// TIA Portal V17 export
// export: Created 2023-02-13T11:16:32.2818041Z, ExportSetting WithDefaults, DisplayName Totally Integrated Automation Portal, DisplayVersion V17, DisplayName TIA Portal Openness, DisplayVersion V17, DisplayName TIA Portal Teamcenter Gateway, DisplayVersion V17, DisplayName TIA Portal Version Control Interface, DisplayVersion V17, DisplayName SINAMICS Startdrive Advanced, DisplayVersion V17, DisplayName SINAMICS Startdrive G130, G150, S120, S150, SINAMICS MV, S210, DisplayVersion V17, DisplayName SINAMICS Startdrive G110M, G120, G120C, G120D, G120P, G115D, DisplayVersion V17, DisplayName STEP 7 Professional, DisplayVersion V17, DisplayName STEP 7 Safety, DisplayVersion V17, DisplayName WinCC Professional, DisplayVersion V17
FUNCTION_BLOCK "IO Valve T51 HotWaterLine"   // FB311, LAD
{ S7_Optimized_Access := 'FALSE' }
VERSION : 0.1
// stored: AutoNumber false, IsIECCheckEnabled false, SetENOAutomatically false, UDAEnableTagReadback false
   VAR_INPUT
      lock : Bool;
      Init : Bool;
      testing : Bool;
      Reset : Bool;
   END_VAR
   VAR
      "AV-51.01" { S7_SetPoint := 'True'} : "Valve";
      "AV-51.02" { S7_SetPoint := 'True'} : "Valve";
      "AV-51.03" { S7_SetPoint := 'True'} : "Valve";
      "AV-51.04" { S7_SetPoint := 'True'} : "Valve";
      "AV-51.05" { S7_SetPoint := 'True'} : "Valve";
      "AV-51.06" { S7_SetPoint := 'True'} : "Valve";
      "AV-51.07" { S7_SetPoint := 'True'} : "Valve";
      "AV-51.08" { S7_SetPoint := 'True'} : "Valve";
      "AV-51.09" { S7_SetPoint := 'True'} : "Valve";
      "AV-51.10" { S7_SetPoint := 'True'} : "Valve";
      "AV-51.11" { S7_SetPoint := 'True'} : "Valve";
      "AV-51.12" { S7_SetPoint := 'True'} : "Valve";
      "AV-51.13" { S7_SetPoint := 'True'} : "Valve";
      "AV-51.14" { S7_SetPoint := 'True'} : "Valve";
      "AV-51.15" { S7_SetPoint := 'True'} : "Valve";
      "CV-51.11" { S7_SetPoint := 'True'} : "Valve";
   END_VAR
BEGIN

REGION Network 1 (SCL): FB OPEN and CLOSE
   IF #testing THEN
       // Statement section IF
       #"AV-51.01".FB_OPEN := #"AV-51.01".QCMD_OP;
       #"AV-51.01".FB_CLOSE := NOT #"AV-51.01".QCMD_OP;
       #"AV-51.02".FB_OPEN := #"AV-51.02".QCMD_OP;
       #"AV-51.02".FB_CLOSE := NOT #"AV-51.02".QCMD_OP;
       #"AV-51.03".FB_OPEN := #"AV-51.03".QCMD_OP;
       #"AV-51.03".FB_CLOSE := NOT #"AV-51.03".QCMD_OP;
       #"AV-51.04".FB_OPEN := #"AV-51.04".QCMD_OP;
       #"AV-51.04".FB_CLOSE := NOT #"AV-51.04".QCMD_OP;
       #"AV-51.05".FB_OPEN := #"AV-51.05".QCMD_OP;
       #"AV-51.05".FB_CLOSE := NOT #"AV-51.05".QCMD_OP;
       #"AV-51.06".FB_OPEN := #"AV-51.06".QCMD_OP;
       #"AV-51.06".FB_CLOSE := NOT #"AV-51.06".QCMD_OP;
       #"AV-51.07".FB_OPEN := #"AV-51.07".QCMD_OP;
       #"AV-51.07".FB_CLOSE := NOT #"AV-51.07".QCMD_OP;
       #"AV-51.08".FB_OPEN := #"AV-51.08".QCMD_OP;
       #"AV-51.08".FB_CLOSE := NOT #"AV-51.08".QCMD_OP;
       #"AV-51.09".FB_OPEN := #"AV-51.09".QCMD_OP;
       #"AV-51.09".FB_CLOSE := NOT #"AV-51.09".QCMD_OP;
       #"AV-51.10".FB_OPEN := #"AV-51.10".QCMD_OP;
       #"AV-51.10".FB_CLOSE := NOT #"AV-51.10".QCMD_OP;
       #"AV-51.11".FB_OPEN := #"AV-51.11".QCMD_OP;
       #"AV-51.11".FB_CLOSE := NOT #"AV-51.11".QCMD_OP;
       #"AV-51.12".FB_OPEN := #"AV-51.12".QCMD_OP;
       #"AV-51.12".FB_CLOSE := NOT #"AV-51.12".QCMD_OP;
       #"AV-51.13".FB_OPEN := #"AV-51.13".QCMD_OP;
       #"AV-51.13".FB_CLOSE := NOT #"AV-51.13".QCMD_OP;
       #"AV-51.14".FB_OPEN := #"AV-51.14".QCMD_OP;
       #"AV-51.14".FB_CLOSE := NOT #"AV-51.14".QCMD_OP;
       #"AV-51.15".FB_OPEN := #"AV-51.15".QCMD_OP;
       #"AV-51.15".FB_CLOSE := NOT #"AV-51.15".QCMD_OP;
   ELSE
       // Statement section ELSE
       #"AV-51.01".FB_OPEN := #"AV-51.01".QCMD_OP;
       #"AV-51.01".FB_CLOSE := NOT #"AV-51.01".QCMD_OP;
       #"AV-51.02".FB_OPEN := #"AV-51.02".QCMD_OP;
       #"AV-51.02".FB_CLOSE := NOT #"AV-51.02".QCMD_OP;
       #"AV-51.03".FB_OPEN := #"AV-51.03".QCMD_OP;
       #"AV-51.03".FB_CLOSE := NOT #"AV-51.03".QCMD_OP;
       #"AV-51.04".FB_OPEN := NOT "ZSC-51.04";
       #"AV-51.04".FB_CLOSE := "ZSC-51.04";
       #"AV-51.05".FB_OPEN := NOT "ZSC-51.05";
       #"AV-51.05".FB_CLOSE := "ZSC-51.05";
       #"AV-51.06".FB_OPEN := #"AV-51.06".QCMD_OP;
       #"AV-51.06".FB_CLOSE := NOT #"AV-51.06".QCMD_OP;
       #"AV-51.07".FB_OPEN := #"AV-51.07".QCMD_OP;
       #"AV-51.07".FB_CLOSE := NOT #"AV-51.07".QCMD_OP;
       #"AV-51.08".FB_OPEN := #"AV-51.08".QCMD_OP;
       #"AV-51.08".FB_CLOSE := NOT #"AV-51.08".QCMD_OP;
       #"AV-51.09".FB_OPEN := #"AV-51.09".QCMD_OP;
       #"AV-51.09".FB_CLOSE := NOT #"AV-51.09".QCMD_OP;
       #"AV-51.10".FB_OPEN := #"AV-51.10".QCMD_OP;
       #"AV-51.10".FB_CLOSE := NOT #"AV-51.10".QCMD_OP;
       #"AV-51.11".FB_OPEN := #"AV-51.11".QCMD_OP;
       #"AV-51.11".FB_CLOSE := NOT #"AV-51.11".QCMD_OP;
       #"AV-51.12".FB_OPEN := #"AV-51.12".QCMD_OP;
       #"AV-51.12".FB_CLOSE := NOT #"AV-51.12".QCMD_OP;
       #"AV-51.13".FB_OPEN := #"AV-51.13".QCMD_OP;
       #"AV-51.13".FB_CLOSE := NOT #"AV-51.13".QCMD_OP;
       #"AV-51.14".FB_OPEN := #"AV-51.14".QCMD_OP;
       #"AV-51.14".FB_CLOSE := NOT #"AV-51.14".QCMD_OP;
       #"AV-51.15".FB_OPEN := #"AV-51.15".QCMD_OP;
       #"AV-51.15".FB_CLOSE := NOT #"AV-51.15".QCMD_OP;
   END_IF;
END_REGION

NETWORK
TITLE = FB Monitoring Time
// FB OPEN Time
      L     t#20s;
      T     #"AV-51.01".MON_T;
      T     #"AV-51.02".MON_T;
      T     #"AV-51.03".MON_T;
      T     #"AV-51.04".MON_T;
      T     #"AV-51.05".MON_T;
      T     #"AV-51.06".MON_T;
      T     #"AV-51.07".MON_T;
      T     #"AV-51.08".MON_T;
      T     #"AV-51.09".MON_T;
      T     #"AV-51.10".MON_T;
      T     #"AV-51.11".MON_T;
      T     #"AV-51.12".MON_T;
      T     #"AV-51.13".MON_T;
      T     #"AV-51.14".MON_T;
      T     #"AV-51.15".MON_T;
// FB CLOSE Time
      L     t#20s;
      T     #"AV-51.01".MON_T_CLOSE;
      T     #"AV-51.02".MON_T_CLOSE;
      T     #"AV-51.03".MON_T_CLOSE;
      T     #"AV-51.04".MON_T_CLOSE;
      T     #"AV-51.05".MON_T_CLOSE;
      T     #"AV-51.06".MON_T_CLOSE;
      T     #"AV-51.07".MON_T_CLOSE;
      T     #"AV-51.08".MON_T_CLOSE;
      T     #"AV-51.09".MON_T_CLOSE;
      T     #"AV-51.10".MON_T_CLOSE;
      T     #"AV-51.11".MON_T_CLOSE;
      T     #"AV-51.12".MON_T_CLOSE;
      T     #"AV-51.13".MON_T_CLOSE;
      T     #"AV-51.14".MON_T_CLOSE;
      T     #"AV-51.15".MON_T_CLOSE;

REGION Network 3: AV-51.01
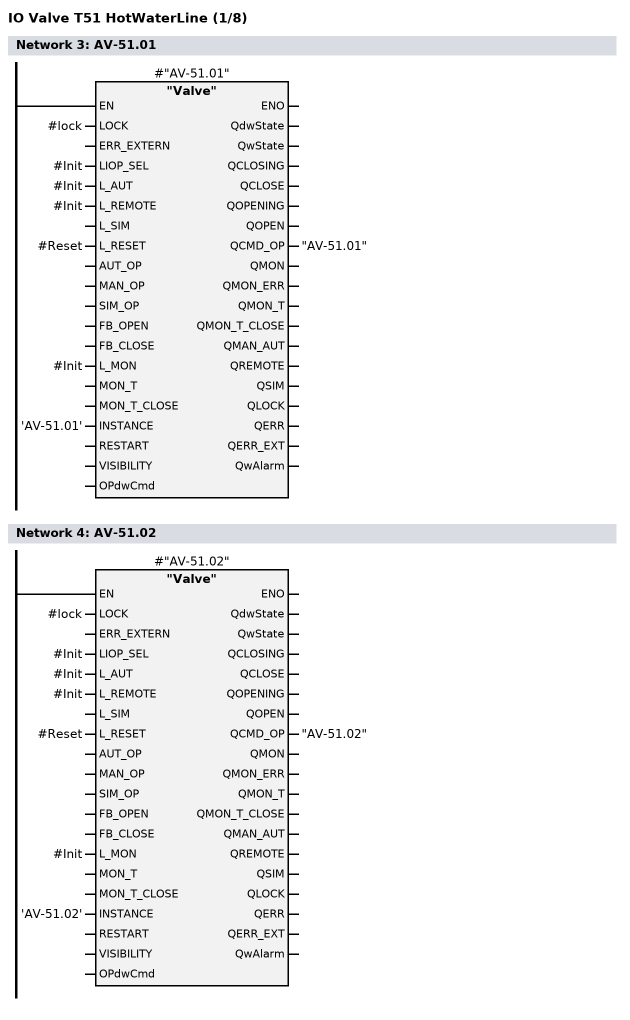
   RUNG wire#powerrail
      #"AV-51.01"(LOCK := #lock, ERR_EXTERN :=, LIOP_SEL := #Init, L_AUT := #Init, L_REMOTE := #Init, L_SIM :=, L_RESET := #Reset, AUT_OP :=, MAN_OP :=, SIM_OP :=, FB_OPEN :=, FB_CLOSE :=, L_MON := #Init, MON_T :=, MON_T_CLOSE :=, INSTANCE := 'AV-51.01', RESTART :=, VISIBILITY :=, OPdwCmd :=, QdwState =>, QwState =>, QCLOSING =>, QCLOSE =>, QOPENING =>, QOPEN =>, QCMD_OP => "AV-51.01", QMON =>, QMON_ERR =>, QMON_T =>, QMON_T_CLOSE =>, QMAN_AUT =>, QREMOTE =>, QSIM =>, QLOCK =>, QERR =>, QERR_EXT =>, QwAlarm =>)
   END_RUNG
   // the same network as SCL:
   #"AV-51.01"(LOCK := #lock,   // "Valve"
               LIOP_SEL := #Init,
               L_AUT := #Init,
               L_REMOTE := #Init,
               L_RESET := #Reset,
               L_MON := #Init,
               INSTANCE := 'AV-51.01',
               QCMD_OP => "AV-51.01");
END_REGION

REGION Network 4: AV-51.02
   RUNG wire#powerrail
      #"AV-51.02"(LOCK := #lock, ERR_EXTERN :=, LIOP_SEL := #Init, L_AUT := #Init, L_REMOTE := #Init, L_SIM :=, L_RESET := #Reset, AUT_OP :=, MAN_OP :=, SIM_OP :=, FB_OPEN :=, FB_CLOSE :=, L_MON := #Init, MON_T :=, MON_T_CLOSE :=, INSTANCE := 'AV-51.02', RESTART :=, VISIBILITY :=, OPdwCmd :=, QdwState =>, QwState =>, QCLOSING =>, QCLOSE =>, QOPENING =>, QOPEN =>, QCMD_OP => "AV-51.02", QMON =>, QMON_ERR =>, QMON_T =>, QMON_T_CLOSE =>, QMAN_AUT =>, QREMOTE =>, QSIM =>, QLOCK =>, QERR =>, QERR_EXT =>, QwAlarm =>)
   END_RUNG
   // the same network as SCL:
   #"AV-51.02"(LOCK := #lock,   // "Valve"
               LIOP_SEL := #Init,
               L_AUT := #Init,
               L_REMOTE := #Init,
               L_RESET := #Reset,
               L_MON := #Init,
               INSTANCE := 'AV-51.02',
               QCMD_OP => "AV-51.02");
END_REGION

REGION Network 5: AV-51.03
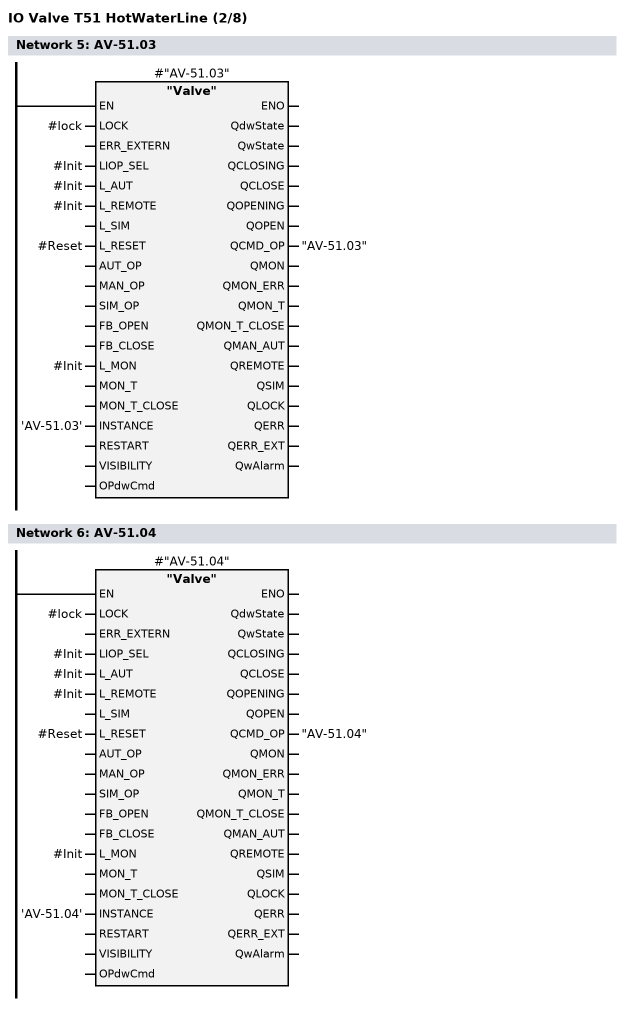
   RUNG wire#powerrail
      #"AV-51.03"(LOCK := #lock, ERR_EXTERN :=, LIOP_SEL := #Init, L_AUT := #Init, L_REMOTE := #Init, L_SIM :=, L_RESET := #Reset, AUT_OP :=, MAN_OP :=, SIM_OP :=, FB_OPEN :=, FB_CLOSE :=, L_MON := #Init, MON_T :=, MON_T_CLOSE :=, INSTANCE := 'AV-51.03', RESTART :=, VISIBILITY :=, OPdwCmd :=, QdwState =>, QwState =>, QCLOSING =>, QCLOSE =>, QOPENING =>, QOPEN =>, QCMD_OP => "AV-51.03", QMON =>, QMON_ERR =>, QMON_T =>, QMON_T_CLOSE =>, QMAN_AUT =>, QREMOTE =>, QSIM =>, QLOCK =>, QERR =>, QERR_EXT =>, QwAlarm =>)
   END_RUNG
   // the same network as SCL:
   #"AV-51.03"(LOCK := #lock,   // "Valve"
               LIOP_SEL := #Init,
               L_AUT := #Init,
               L_REMOTE := #Init,
               L_RESET := #Reset,
               L_MON := #Init,
               INSTANCE := 'AV-51.03',
               QCMD_OP => "AV-51.03");
END_REGION

REGION Network 6: AV-51.04
   RUNG wire#powerrail
      #"AV-51.04"(LOCK := #lock, ERR_EXTERN :=, LIOP_SEL := #Init, L_AUT := #Init, L_REMOTE := #Init, L_SIM :=, L_RESET := #Reset, AUT_OP :=, MAN_OP :=, SIM_OP :=, FB_OPEN :=, FB_CLOSE :=, L_MON := #Init, MON_T :=, MON_T_CLOSE :=, INSTANCE := 'AV-51.04', RESTART :=, VISIBILITY :=, OPdwCmd :=, QdwState =>, QwState =>, QCLOSING =>, QCLOSE =>, QOPENING =>, QOPEN =>, QCMD_OP => "AV-51.04", QMON =>, QMON_ERR =>, QMON_T =>, QMON_T_CLOSE =>, QMAN_AUT =>, QREMOTE =>, QSIM =>, QLOCK =>, QERR =>, QERR_EXT =>, QwAlarm =>)
   END_RUNG
   // the same network as SCL:
   #"AV-51.04"(LOCK := #lock,   // "Valve"
               LIOP_SEL := #Init,
               L_AUT := #Init,
               L_REMOTE := #Init,
               L_RESET := #Reset,
               L_MON := #Init,
               INSTANCE := 'AV-51.04',
               QCMD_OP => "AV-51.04");
END_REGION

REGION Network 7: AV-51.05
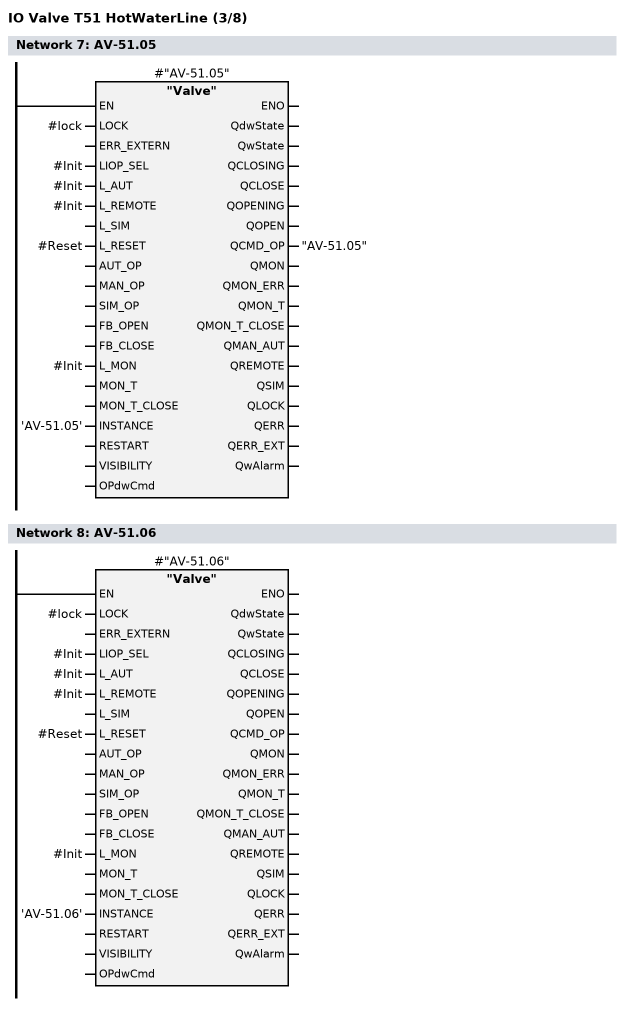
   RUNG wire#powerrail
      #"AV-51.05"(LOCK := #lock, ERR_EXTERN :=, LIOP_SEL := #Init, L_AUT := #Init, L_REMOTE := #Init, L_SIM :=, L_RESET := #Reset, AUT_OP :=, MAN_OP :=, SIM_OP :=, FB_OPEN :=, FB_CLOSE :=, L_MON := #Init, MON_T :=, MON_T_CLOSE :=, INSTANCE := 'AV-51.05', RESTART :=, VISIBILITY :=, OPdwCmd :=, QdwState =>, QwState =>, QCLOSING =>, QCLOSE =>, QOPENING =>, QOPEN =>, QCMD_OP => "AV-51.05", QMON =>, QMON_ERR =>, QMON_T =>, QMON_T_CLOSE =>, QMAN_AUT =>, QREMOTE =>, QSIM =>, QLOCK =>, QERR =>, QERR_EXT =>, QwAlarm =>)
   END_RUNG
   // the same network as SCL:
   #"AV-51.05"(LOCK := #lock,   // "Valve"
               LIOP_SEL := #Init,
               L_AUT := #Init,
               L_REMOTE := #Init,
               L_RESET := #Reset,
               L_MON := #Init,
               INSTANCE := 'AV-51.05',
               QCMD_OP => "AV-51.05");
END_REGION

REGION Network 8: AV-51.06
   RUNG wire#powerrail
      #"AV-51.06"(LOCK := #lock, ERR_EXTERN :=, LIOP_SEL := #Init, L_AUT := #Init, L_REMOTE := #Init, L_SIM :=, L_RESET := #Reset, AUT_OP :=, MAN_OP :=, SIM_OP :=, FB_OPEN :=, FB_CLOSE :=, L_MON := #Init, MON_T :=, MON_T_CLOSE :=, INSTANCE := 'AV-51.06', RESTART :=, VISIBILITY :=, OPdwCmd :=, QdwState =>, QwState =>, QCLOSING =>, QCLOSE =>, QOPENING =>, QOPEN =>, QCMD_OP =>, QMON =>, QMON_ERR =>, QMON_T =>, QMON_T_CLOSE =>, QMAN_AUT =>, QREMOTE =>, QSIM =>, QLOCK =>, QERR =>, QERR_EXT =>, QwAlarm =>)
   END_RUNG
   // the same network as SCL:
   #"AV-51.06"(LOCK := #lock,   // "Valve"
               LIOP_SEL := #Init,
               L_AUT := #Init,
               L_REMOTE := #Init,
               L_RESET := #Reset,
               L_MON := #Init,
               INSTANCE := 'AV-51.06');
END_REGION

REGION Network 9: AV-51.07
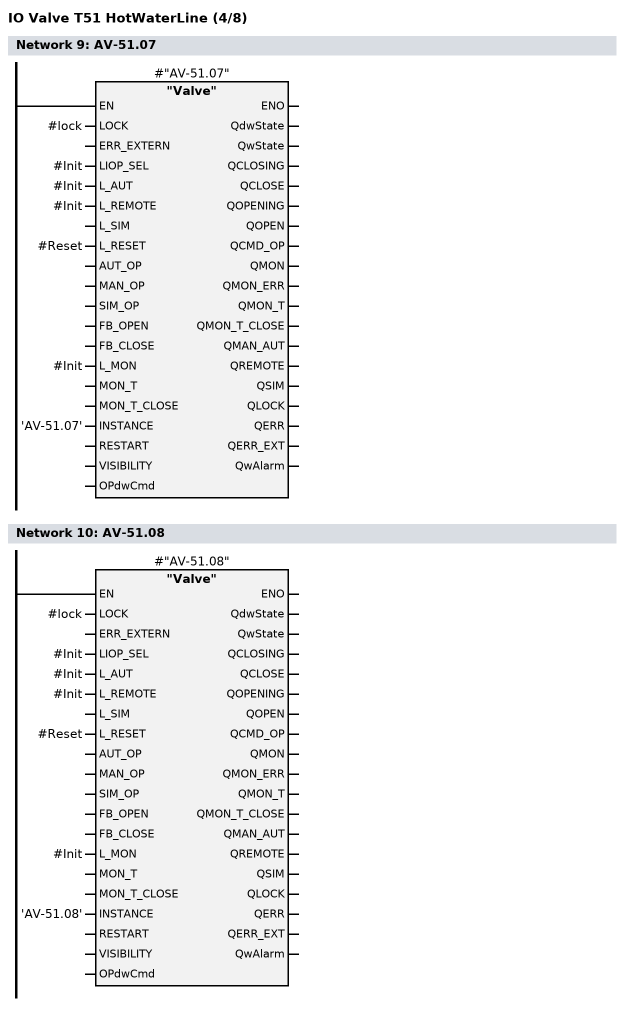
   RUNG wire#powerrail
      #"AV-51.07"(LOCK := #lock, ERR_EXTERN :=, LIOP_SEL := #Init, L_AUT := #Init, L_REMOTE := #Init, L_SIM :=, L_RESET := #Reset, AUT_OP :=, MAN_OP :=, SIM_OP :=, FB_OPEN :=, FB_CLOSE :=, L_MON := #Init, MON_T :=, MON_T_CLOSE :=, INSTANCE := 'AV-51.07', RESTART :=, VISIBILITY :=, OPdwCmd :=, QdwState =>, QwState =>, QCLOSING =>, QCLOSE =>, QOPENING =>, QOPEN =>, QCMD_OP =>, QMON =>, QMON_ERR =>, QMON_T =>, QMON_T_CLOSE =>, QMAN_AUT =>, QREMOTE =>, QSIM =>, QLOCK =>, QERR =>, QERR_EXT =>, QwAlarm =>)
   END_RUNG
   // the same network as SCL:
   #"AV-51.07"(LOCK := #lock,   // "Valve"
               LIOP_SEL := #Init,
               L_AUT := #Init,
               L_REMOTE := #Init,
               L_RESET := #Reset,
               L_MON := #Init,
               INSTANCE := 'AV-51.07');
END_REGION

REGION Network 10: AV-51.08
   RUNG wire#powerrail
      #"AV-51.08"(LOCK := #lock, ERR_EXTERN :=, LIOP_SEL := #Init, L_AUT := #Init, L_REMOTE := #Init, L_SIM :=, L_RESET := #Reset, AUT_OP :=, MAN_OP :=, SIM_OP :=, FB_OPEN :=, FB_CLOSE :=, L_MON := #Init, MON_T :=, MON_T_CLOSE :=, INSTANCE := 'AV-51.08', RESTART :=, VISIBILITY :=, OPdwCmd :=, QdwState =>, QwState =>, QCLOSING =>, QCLOSE =>, QOPENING =>, QOPEN =>, QCMD_OP =>, QMON =>, QMON_ERR =>, QMON_T =>, QMON_T_CLOSE =>, QMAN_AUT =>, QREMOTE =>, QSIM =>, QLOCK =>, QERR =>, QERR_EXT =>, QwAlarm =>)
   END_RUNG
   // the same network as SCL:
   #"AV-51.08"(LOCK := #lock,   // "Valve"
               LIOP_SEL := #Init,
               L_AUT := #Init,
               L_REMOTE := #Init,
               L_RESET := #Reset,
               L_MON := #Init,
               INSTANCE := 'AV-51.08');
END_REGION

REGION Network 11: AV-51.09
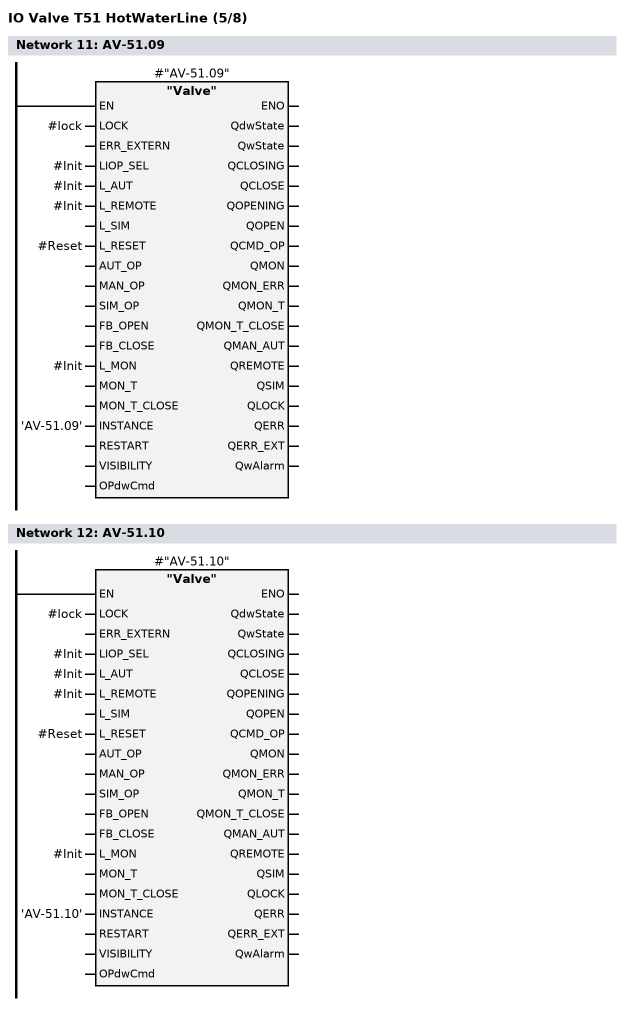
   RUNG wire#powerrail
      #"AV-51.09"(LOCK := #lock, ERR_EXTERN :=, LIOP_SEL := #Init, L_AUT := #Init, L_REMOTE := #Init, L_SIM :=, L_RESET := #Reset, AUT_OP :=, MAN_OP :=, SIM_OP :=, FB_OPEN :=, FB_CLOSE :=, L_MON := #Init, MON_T :=, MON_T_CLOSE :=, INSTANCE := 'AV-51.09', RESTART :=, VISIBILITY :=, OPdwCmd :=, QdwState =>, QwState =>, QCLOSING =>, QCLOSE =>, QOPENING =>, QOPEN =>, QCMD_OP =>, QMON =>, QMON_ERR =>, QMON_T =>, QMON_T_CLOSE =>, QMAN_AUT =>, QREMOTE =>, QSIM =>, QLOCK =>, QERR =>, QERR_EXT =>, QwAlarm =>)
   END_RUNG
   // the same network as SCL:
   #"AV-51.09"(LOCK := #lock,   // "Valve"
               LIOP_SEL := #Init,
               L_AUT := #Init,
               L_REMOTE := #Init,
               L_RESET := #Reset,
               L_MON := #Init,
               INSTANCE := 'AV-51.09');
END_REGION

REGION Network 12: AV-51.10
   RUNG wire#powerrail
      #"AV-51.10"(LOCK := #lock, ERR_EXTERN :=, LIOP_SEL := #Init, L_AUT := #Init, L_REMOTE := #Init, L_SIM :=, L_RESET := #Reset, AUT_OP :=, MAN_OP :=, SIM_OP :=, FB_OPEN :=, FB_CLOSE :=, L_MON := #Init, MON_T :=, MON_T_CLOSE :=, INSTANCE := 'AV-51.10', RESTART :=, VISIBILITY :=, OPdwCmd :=, QdwState =>, QwState =>, QCLOSING =>, QCLOSE =>, QOPENING =>, QOPEN =>, QCMD_OP =>, QMON =>, QMON_ERR =>, QMON_T =>, QMON_T_CLOSE =>, QMAN_AUT =>, QREMOTE =>, QSIM =>, QLOCK =>, QERR =>, QERR_EXT =>, QwAlarm =>)
   END_RUNG
   // the same network as SCL:
   #"AV-51.10"(LOCK := #lock,   // "Valve"
               LIOP_SEL := #Init,
               L_AUT := #Init,
               L_REMOTE := #Init,
               L_RESET := #Reset,
               L_MON := #Init,
               INSTANCE := 'AV-51.10');
END_REGION

REGION Network 13: AV-51.11
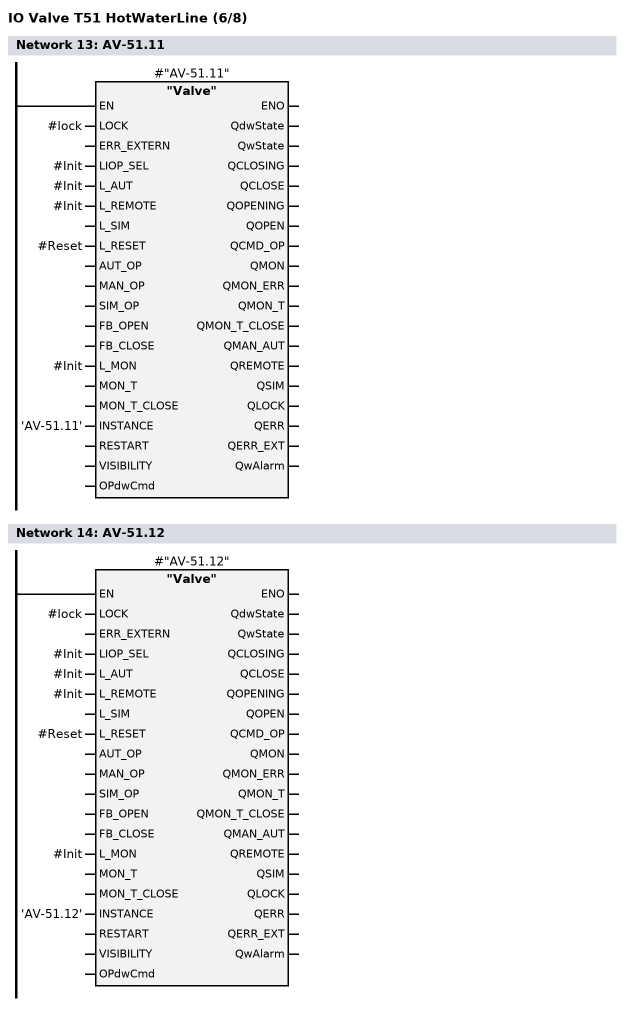
   RUNG wire#powerrail
      #"AV-51.11"(LOCK := #lock, ERR_EXTERN :=, LIOP_SEL := #Init, L_AUT := #Init, L_REMOTE := #Init, L_SIM :=, L_RESET := #Reset, AUT_OP :=, MAN_OP :=, SIM_OP :=, FB_OPEN :=, FB_CLOSE :=, L_MON := #Init, MON_T :=, MON_T_CLOSE :=, INSTANCE := 'AV-51.11', RESTART :=, VISIBILITY :=, OPdwCmd :=, QdwState =>, QwState =>, QCLOSING =>, QCLOSE =>, QOPENING =>, QOPEN =>, QCMD_OP =>, QMON =>, QMON_ERR =>, QMON_T =>, QMON_T_CLOSE =>, QMAN_AUT =>, QREMOTE =>, QSIM =>, QLOCK =>, QERR =>, QERR_EXT =>, QwAlarm =>)
   END_RUNG
   // the same network as SCL:
   #"AV-51.11"(LOCK := #lock,   // "Valve"
               LIOP_SEL := #Init,
               L_AUT := #Init,
               L_REMOTE := #Init,
               L_RESET := #Reset,
               L_MON := #Init,
               INSTANCE := 'AV-51.11');
END_REGION

REGION Network 14: AV-51.12
   RUNG wire#powerrail
      #"AV-51.12"(LOCK := #lock, ERR_EXTERN :=, LIOP_SEL := #Init, L_AUT := #Init, L_REMOTE := #Init, L_SIM :=, L_RESET := #Reset, AUT_OP :=, MAN_OP :=, SIM_OP :=, FB_OPEN :=, FB_CLOSE :=, L_MON := #Init, MON_T :=, MON_T_CLOSE :=, INSTANCE := 'AV-51.12', RESTART :=, VISIBILITY :=, OPdwCmd :=, QdwState =>, QwState =>, QCLOSING =>, QCLOSE =>, QOPENING =>, QOPEN =>, QCMD_OP =>, QMON =>, QMON_ERR =>, QMON_T =>, QMON_T_CLOSE =>, QMAN_AUT =>, QREMOTE =>, QSIM =>, QLOCK =>, QERR =>, QERR_EXT =>, QwAlarm =>)
   END_RUNG
   // the same network as SCL:
   #"AV-51.12"(LOCK := #lock,   // "Valve"
               LIOP_SEL := #Init,
               L_AUT := #Init,
               L_REMOTE := #Init,
               L_RESET := #Reset,
               L_MON := #Init,
               INSTANCE := 'AV-51.12');
END_REGION

REGION Network 15: AV-51.13
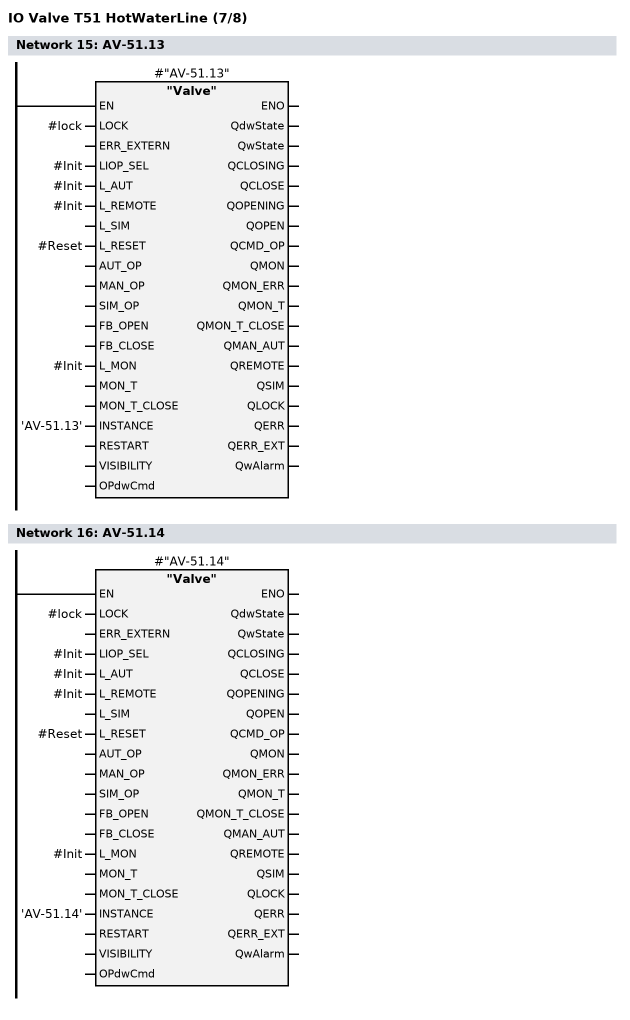
   RUNG wire#powerrail
      #"AV-51.13"(LOCK := #lock, ERR_EXTERN :=, LIOP_SEL := #Init, L_AUT := #Init, L_REMOTE := #Init, L_SIM :=, L_RESET := #Reset, AUT_OP :=, MAN_OP :=, SIM_OP :=, FB_OPEN :=, FB_CLOSE :=, L_MON := #Init, MON_T :=, MON_T_CLOSE :=, INSTANCE := 'AV-51.13', RESTART :=, VISIBILITY :=, OPdwCmd :=, QdwState =>, QwState =>, QCLOSING =>, QCLOSE =>, QOPENING =>, QOPEN =>, QCMD_OP =>, QMON =>, QMON_ERR =>, QMON_T =>, QMON_T_CLOSE =>, QMAN_AUT =>, QREMOTE =>, QSIM =>, QLOCK =>, QERR =>, QERR_EXT =>, QwAlarm =>)
   END_RUNG
   // the same network as SCL:
   #"AV-51.13"(LOCK := #lock,   // "Valve"
               LIOP_SEL := #Init,
               L_AUT := #Init,
               L_REMOTE := #Init,
               L_RESET := #Reset,
               L_MON := #Init,
               INSTANCE := 'AV-51.13');
END_REGION

REGION Network 16: AV-51.14
   RUNG wire#powerrail
      #"AV-51.14"(LOCK := #lock, ERR_EXTERN :=, LIOP_SEL := #Init, L_AUT := #Init, L_REMOTE := #Init, L_SIM :=, L_RESET := #Reset, AUT_OP :=, MAN_OP :=, SIM_OP :=, FB_OPEN :=, FB_CLOSE :=, L_MON := #Init, MON_T :=, MON_T_CLOSE :=, INSTANCE := 'AV-51.14', RESTART :=, VISIBILITY :=, OPdwCmd :=, QdwState =>, QwState =>, QCLOSING =>, QCLOSE =>, QOPENING =>, QOPEN =>, QCMD_OP =>, QMON =>, QMON_ERR =>, QMON_T =>, QMON_T_CLOSE =>, QMAN_AUT =>, QREMOTE =>, QSIM =>, QLOCK =>, QERR =>, QERR_EXT =>, QwAlarm =>)
   END_RUNG
   // the same network as SCL:
   #"AV-51.14"(LOCK := #lock,   // "Valve"
               LIOP_SEL := #Init,
               L_AUT := #Init,
               L_REMOTE := #Init,
               L_RESET := #Reset,
               L_MON := #Init,
               INSTANCE := 'AV-51.14');
END_REGION

REGION Network 17: AV-51.15
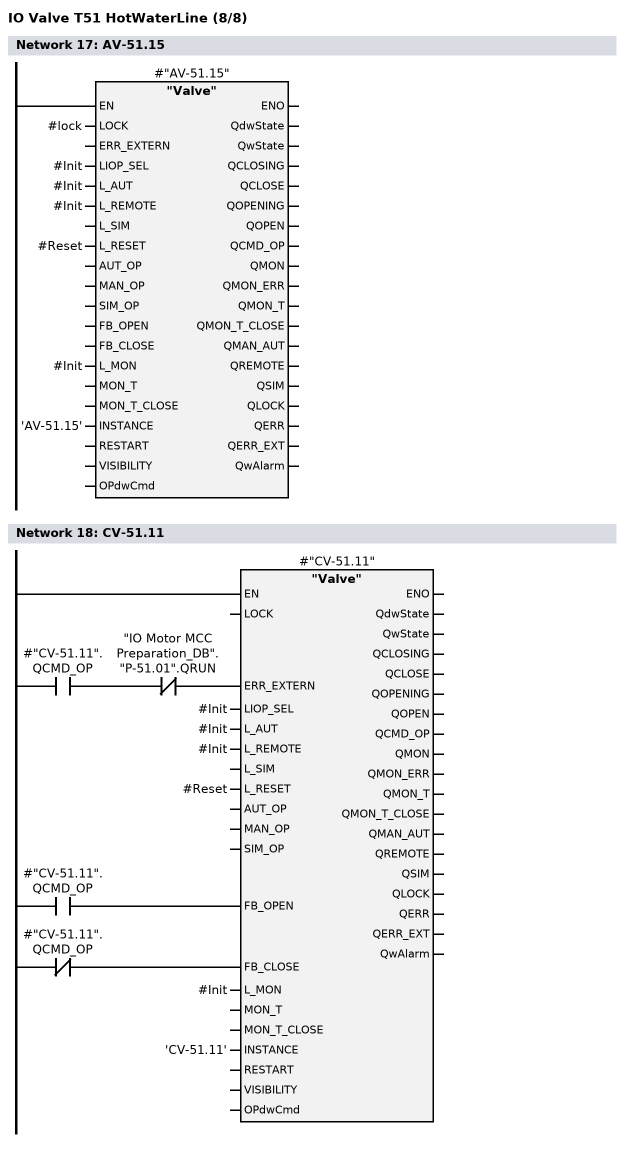
   RUNG wire#powerrail
      #"AV-51.15"(LOCK := #lock, ERR_EXTERN :=, LIOP_SEL := #Init, L_AUT := #Init, L_REMOTE := #Init, L_SIM :=, L_RESET := #Reset, AUT_OP :=, MAN_OP :=, SIM_OP :=, FB_OPEN :=, FB_CLOSE :=, L_MON := #Init, MON_T :=, MON_T_CLOSE :=, INSTANCE := 'AV-51.15', RESTART :=, VISIBILITY :=, OPdwCmd :=, QdwState =>, QwState =>, QCLOSING =>, QCLOSE =>, QOPENING =>, QOPEN =>, QCMD_OP =>, QMON =>, QMON_ERR =>, QMON_T =>, QMON_T_CLOSE =>, QMAN_AUT =>, QREMOTE =>, QSIM =>, QLOCK =>, QERR =>, QERR_EXT =>, QwAlarm =>)
   END_RUNG
   // the same network as SCL:
   #"AV-51.15"(LOCK := #lock,   // "Valve"
               LIOP_SEL := #Init,
               L_AUT := #Init,
               L_REMOTE := #Init,
               L_RESET := #Reset,
               L_MON := #Init,
               INSTANCE := 'AV-51.15');
END_REGION

REGION Network 18: CV-51.11
   RUNG wire#powerrail
      #"CV-51.11"(ERR_EXTERN := wire#w1, FB_OPEN := wire#w2, FB_CLOSE := wire#w3, LOCK :=, LIOP_SEL := #Init, L_AUT := #Init, L_REMOTE := #Init, L_SIM :=, L_RESET := #Reset, AUT_OP :=, MAN_OP :=, SIM_OP :=, L_MON := #Init, MON_T :=, MON_T_CLOSE :=, INSTANCE := 'CV-51.11', RESTART :=, VISIBILITY :=, OPdwCmd :=, QdwState =>, QwState =>, QCLOSING =>, QCLOSE =>, QOPENING =>, QOPEN =>, QCMD_OP =>, QMON =>, QMON_ERR =>, QMON_T =>, QMON_T_CLOSE =>, QMAN_AUT =>, QREMOTE =>, QSIM =>, QLOCK =>, QERR =>, QERR_EXT =>, QwAlarm =>)
   END_RUNG
   RUNG wire#powerrail
      Contact( #"CV-51.11".QCMD_OP )
      I_Contact( "IO Motor MCC Preparation_DB"."P-51.01".QRUN )
   END_RUNG wire#w1
   RUNG wire#powerrail
      Contact( #"CV-51.11".QCMD_OP )
   END_RUNG wire#w2
   RUNG wire#powerrail
      I_Contact( #"CV-51.11".QCMD_OP )
   END_RUNG wire#w3
   // the same network as SCL:
   #"CV-51.11"(ERR_EXTERN := #"CV-51.11".QCMD_OP AND NOT "IO Motor MCC Preparation_DB"."P-51.01".QRUN,   // "Valve"
               LIOP_SEL := #Init,
               L_AUT := #Init,
               L_REMOTE := #Init,
               L_RESET := #Reset,
               FB_OPEN := #"CV-51.11".QCMD_OP,
               FB_CLOSE := NOT #"CV-51.11".QCMD_OP,
               L_MON := #Init,
               INSTANCE := 'CV-51.11');
END_REGION
END_FUNCTION_BLOCK
